(* Logix 5000 project; controller PLCbox vendor 1 type 14 code 149 rev 30.11; software revision 30.01; part 2 of 3 *)
(* tags used below, declared in another part *)
   HMI_Int_BOOL : BOOL[64];
   Light1_Complete_ONS : BOOL;
   Light1_Green : BOOL;
   Light1_Green_T : TIMER;
   Light1_Red : BOOL;
   Light1_Reset : BOOL;
   Light1_Yellow : BOOL;
   Light1_Yellow_T : TIMER;
   Light2_Complete_ONS : BOOL;
   Light2_Green : BOOL;
   Light2_Green_T : TIMER;
   Light2_Red : BOOL;
   Light2_Reset : BOOL;
   Light2_Yellow : BOOL;
   Light2_Yellow_T : TIMER;
   PID_Analog_In : REAL[20];
   System_Timer : TIMER[100];
   tagToPi : DINT;

PROGRAM MainProgram2   (* main routine _01_Main *)
VAR
   PID_1001 : PID_ENHANCED := (PVEUMax := 100.0, SPOper := 50.0, SPHLimit := 100.0, RatioProg := 1.0, RatioOper := 1.0, RatioHLimit := 1.0, RatioLLimit := 1.0, CVOper := 100.0, CVEUMax := 100.0, CVHLimit := 100.0, DependIndepend := 1, PGain := 0.1, IGain := 0.001, DGain := 0.001, PVEDerivative := 1, ProgOperReq := 1, RTSTime := 1, CVEU := 100.0, CV := 100.0, CVHAlarm := 1, SP := 50.0, SPPercent := 50.0, E := 50.0, EPercent := 50.0, InitPrimary := 1, WindupHOut := 1, Ratio := 1.0, Auto := 1, DeltaT := 0.1);
   PID_Par_1001 : UDT_PID := (P := 0.1, I := 0.001, D := 0.001, CV := 100.0, SP := 50.0, Auto := 1, Name := 'PID 1001 - Testing CLICK PLC Input');
   SCL_01 : SCALE := (InRawMax := 5000.0, InEUMax := 100.0);
END_VAR

ROUTINE _01_Main   (* ladder *)
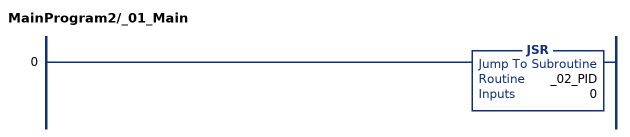
   0: JSR(_02_PID,0);
END_ROUTINE

ROUTINE _02_PID   (* function block diagram *)
   SHEET 1
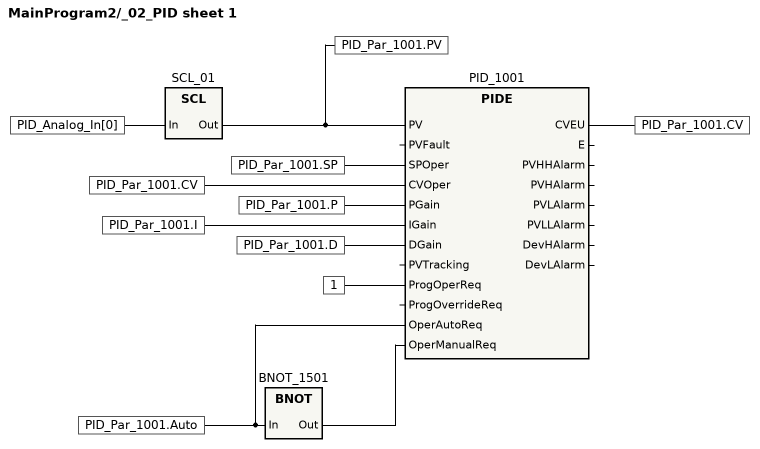
   SCL_01 : SCL(In := PID_Analog_In[0]);
   BNOT_1501 : BNOT(In := PID_Par_1001.Auto);
   PID_Par_1001.PV := SCL_01.Out;
   PID_1001 : PIDE(PV := SCL_01.Out, SPOper := PID_Par_1001.SP, CVOper := PID_Par_1001.CV, PGain := PID_Par_1001.P, IGain := PID_Par_1001.I, DGain := PID_Par_1001.D, ProgOperReq := 1, OperAutoReq := PID_Par_1001.Auto, OperManualReq := BNOT_1501.Out);   // unwired pins: PVFault PVTracking ProgOverrideReq E PVHHAlarm PVHAlarm PVLAlarm PVLLAlarm DevHAlarm DevLAlarm
   PID_Par_1001.CV := PID_1001.CVEU;
END_ROUTINE
END_PROGRAM

PROGRAM Mathematical   (* main routine _01_Main *)
VAR
   System_DINT : DINT[100] := ([0] := 12, [1] := 32, [2] := 54, [3] := 4, [4] := 31, [5] := 38, [6] := 100, [7] := 50, [8] := 200, [9] := 116);
   System_REAL : REAL[100] := ([0] := 23.0, [1] := 42.0, [2] := 0.48835304, [5] := 1.0);
END_VAR

ROUTINE _01_Main   (* ladder *)
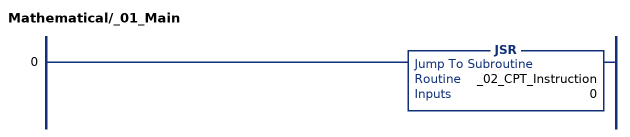
   0: JSR(_02_CPT_Instruction,0);
END_ROUTINE

ROUTINE _02_CPT_Instruction   (* ladder *)
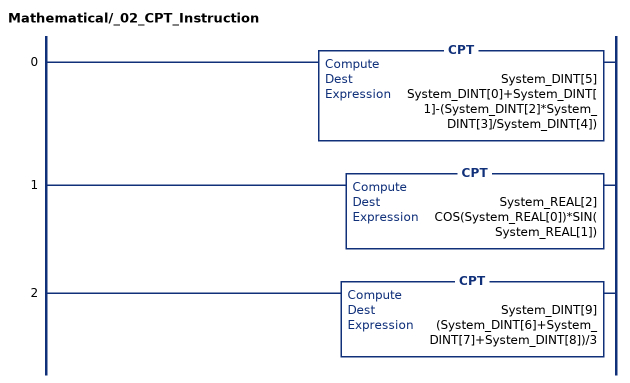
   0: CPT(System_DINT[5],System_DINT[0]+System_DINT[1]-(System_DINT[2]*System_DINT[3]/System_DINT[4]));
   1: CPT(System_REAL[2],COS(System_REAL[0])*SIN(System_REAL[1]));
   2: CPT(System_DINT[9],(System_DINT[6]+System_DINT[7]+System_DINT[8])/3);
END_ROUTINE
END_PROGRAM

PROGRAM PowerFlex525Mastery   (* main routine _01_Main *)
VAR
   Drive_Status : DINT := 1;
   Motor_Dev : REAL := 300.0;
   Motor_Fault_Timer : TIMER := (PRE := 20000);
   Motor_Faulted : BOOL;
   Motor_Run : BOOL;
   Motor_SpdLim_High : REAL := 6300.0;
   Motor_SpdLim_Low : REAL := 5700.0;
   Motor_Target_Speed_Fault : BOOL;
   Reset_PB : BOOL;
   Start_PB : BOOL;
   Stop_PB : BOOL;
END_VAR

ROUTINE _01_Main   (* ladder *)
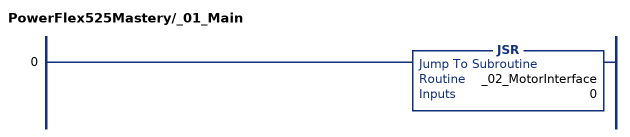
   0: JSR(_02_MotorInterface,0);
END_ROUTINE

ROUTINE _02_MotorInterface   (* ladder *)
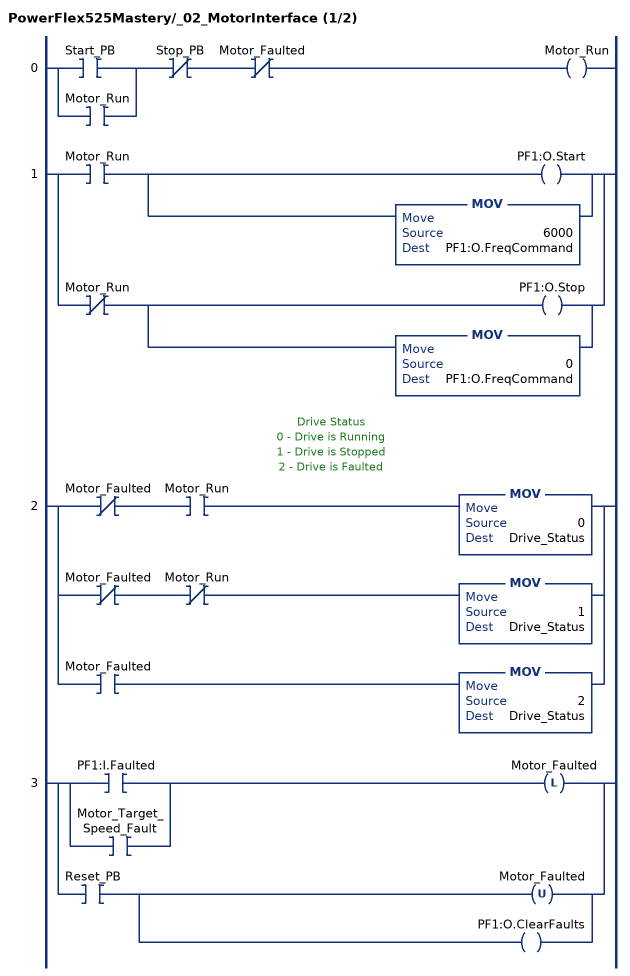
   0: [XIC(Start_PB) ,XIC(Motor_Run) ]XIO(Stop_PB)XIO(Motor_Faulted)OTE(Motor_Run);
   1: [XIC(Motor_Run) [OTE(PF1:O.Start) ,MOV(6000,PF1:O.FreqCommand) ] ,XIO(Motor_Run) [OTE(PF1:O.Stop) ,MOV(0,PF1:O.FreqCommand) ] ];
   // Drive Status
   // 0 - Drive is Running
   // 1 - Drive is Stopped
   // 2 - Drive is Faulted
   2: [XIO(Motor_Faulted) XIC(Motor_Run) MOV(0,Drive_Status) ,XIO(Motor_Faulted) XIO(Motor_Run) MOV(1,Drive_Status) ,XIC(Motor_Faulted) MOV(2,Drive_Status) ];
   3: [[XIC(PF1:I.Faulted) ,XIC(Motor_Target_Speed_Fault) ] OTL(Motor_Faulted) ,XIC(Reset_PB) [OTU(Motor_Faulted) ,OTE(PF1:O.ClearFaults) ] ];
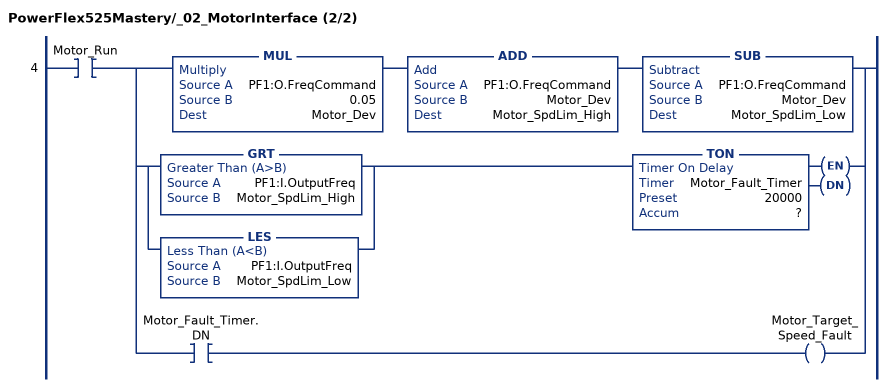
   4: XIC(Motor_Run)[MUL(PF1:O.FreqCommand,0.05,Motor_Dev) ADD(PF1:O.FreqCommand,Motor_Dev,Motor_SpdLim_High) SUB(PF1:O.FreqCommand,Motor_Dev,Motor_SpdLim_Low) ,[GRT(PF1:I.OutputFreq,Motor_SpdLim_High) ,LES(PF1:I.OutputFreq,Motor_SpdLim_Low) ] TON(Motor_Fault_Timer,?,?) ,XIC(Motor_Fault_Timer.DN) OTE(Motor_Target_Speed_Fault) ];
END_ROUTINE
END_PROGRAM

PROGRAM ST_Practice   (* main routine _01_Main *)

ROUTINE _01_Main   (* ladder *)
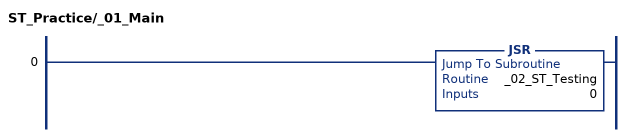
   0: JSR(_02_ST_Testing,0);
END_ROUTINE

ROUTINE _02_ST_Testing   (* structured text *)
   
END_ROUTINE
END_PROGRAM

PROGRAM StreetLightSystem   (* main routine _01_Main *)

ROUTINE _01_Main   (* ladder *)
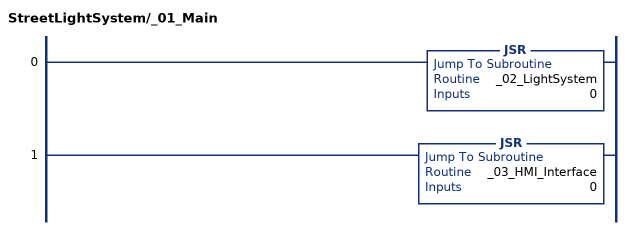
   0: JSR(_02_LightSystem,0);
   1: JSR(_03_HMI_Interface,0);
END_ROUTINE

ROUTINE _02_LightSystem   (* ladder *)
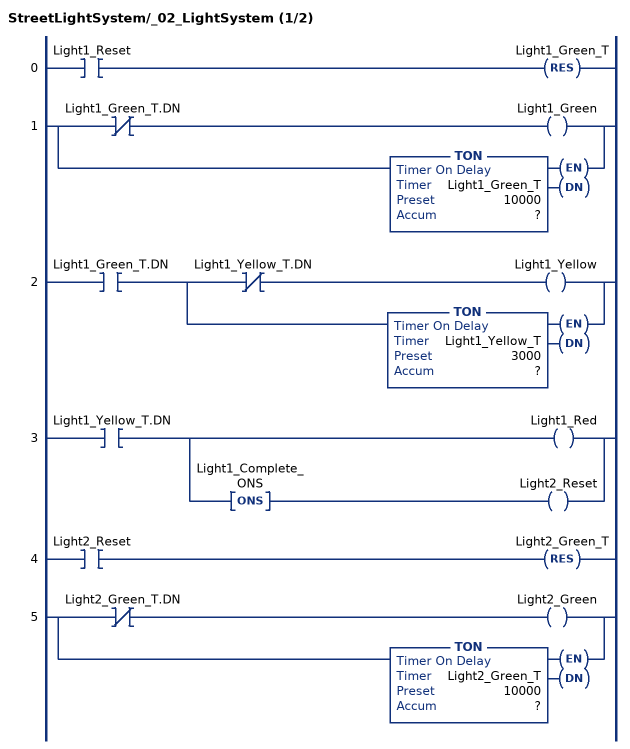
   0: XIC(Light1_Reset)RES(Light1_Green_T);
   1: [XIO(Light1_Green_T.DN) OTE(Light1_Green) ,TON(Light1_Green_T,?,?) ];
   2: XIC(Light1_Green_T.DN)[XIO(Light1_Yellow_T.DN) OTE(Light1_Yellow) ,TON(Light1_Yellow_T,?,?) ];
   3: XIC(Light1_Yellow_T.DN)[OTE(Light1_Red) ,ONS(Light1_Complete_ONS) OTE(Light2_Reset) ];
   4: XIC(Light2_Reset)RES(Light2_Green_T);
   5: [XIO(Light2_Green_T.DN) OTE(Light2_Green) ,TON(Light2_Green_T,?,?) ];
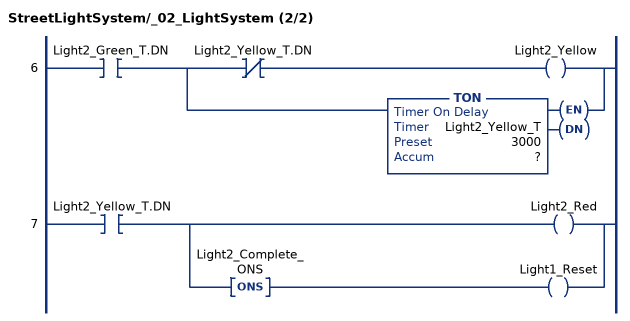
   6: XIC(Light2_Green_T.DN)[XIO(Light2_Yellow_T.DN) OTE(Light2_Yellow) ,TON(Light2_Yellow_T,?,?) ];
   7: XIC(Light2_Yellow_T.DN)[OTE(Light2_Red) ,ONS(Light2_Complete_ONS) OTE(Light1_Reset) ];
END_ROUTINE

ROUTINE _03_HMI_Interface   (* ladder *)
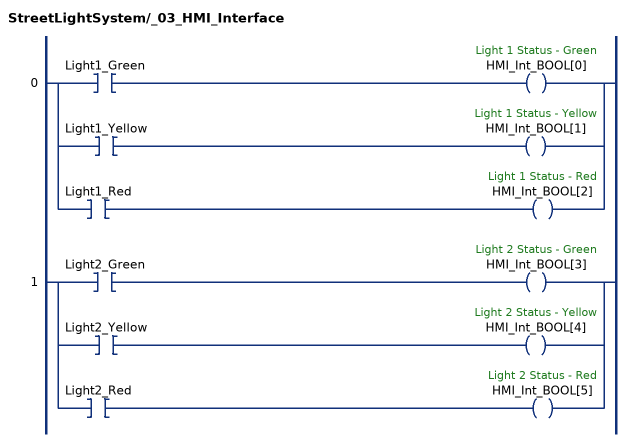
   0: [XIC(Light1_Green) OTE(HMI_Int_BOOL[0]) ,XIC(Light1_Yellow) OTE(HMI_Int_BOOL[1]) ,XIC(Light1_Red) OTE(HMI_Int_BOOL[2]) ];
   1: [XIC(Light2_Green) OTE(HMI_Int_BOOL[3]) ,XIC(Light2_Yellow) OTE(HMI_Int_BOOL[4]) ,XIC(Light2_Red) OTE(HMI_Int_BOOL[5]) ];
END_ROUTINE
END_PROGRAM

PROGRAM TankFillingChallenge   (* main routine _01_Main *)
VAR
   DischargeStatus : DINT := 1;
   FillingStatus : DINT := 1;
   T_Vlad : BOOL[128];
   TankActualLevel : REAL := 42.792046;
   TankDischargeRate : REAL := 0.5;
   TankEmptyThreshold : REAL := 5.0;
   TankFill : BOOL[128];
        [0]   // START Filling Station
        [1]   // STOP Filling Station
        [2]   // Filling Station RUNNING
        [3]   // START Discharge Station
        [4]   // STOP Discharge Station
        [5]   // Discharge Station RUNNING
        [6]   // TANK FULL
        [7]   // TANK EMPTY
   TankFillRate : REAL := 0.3;
   TankFullThreshold : REAL := 100.0;
   TankOut : BOOL[32];
        [0]   // Filling Station VALVE OPEN
        [1]   // Discharge Station VALVE OPEN
   TankTimers : TIMER[10] := ([0].PRE := 20, [1].PRE := 20);
END_VAR

ROUTINE _01_Main   (* ladder *)
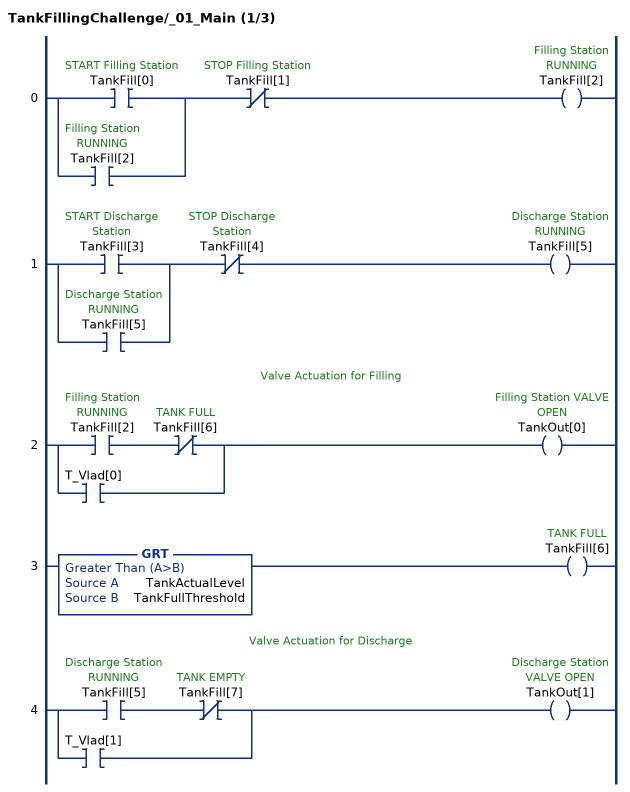
   0: [XIC(TankFill[0]) ,XIC(TankFill[2]) ]XIO(TankFill[1])OTE(TankFill[2]);
   1: [XIC(TankFill[3]) ,XIC(TankFill[5]) ]XIO(TankFill[4])OTE(TankFill[5]);
   // Valve Actuation for Filling
   2: [XIC(TankFill[2]) XIO(TankFill[6]) ,XIC(T_Vlad[0]) ]OTE(TankOut[0]);
   3: GRT(TankActualLevel,TankFullThreshold)OTE(TankFill[6]);
   // Valve Actuation for Discharge
   4: [XIC(TankFill[5]) XIO(TankFill[7]) ,XIC(T_Vlad[1]) ]OTE(TankOut[1]);
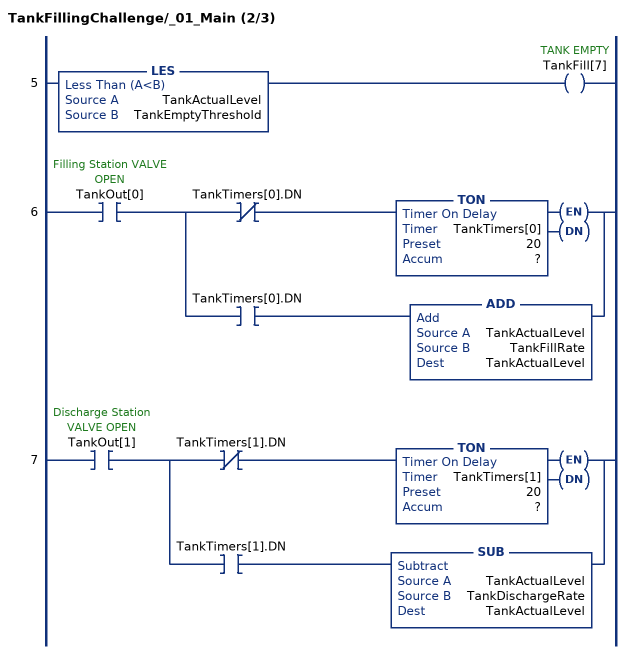
   5: LES(TankActualLevel,TankEmptyThreshold)OTE(TankFill[7]);
   6: XIC(TankOut[0])[XIO(TankTimers[0].DN) TON(TankTimers[0],?,?) ,XIC(TankTimers[0].DN) ADD(TankActualLevel,TankFillRate,TankActualLevel) ];
   7: XIC(TankOut[1])[XIO(TankTimers[1].DN) TON(TankTimers[1],?,?) ,XIC(TankTimers[1].DN) SUB(TankActualLevel,TankDischargeRate,TankActualLevel) ];
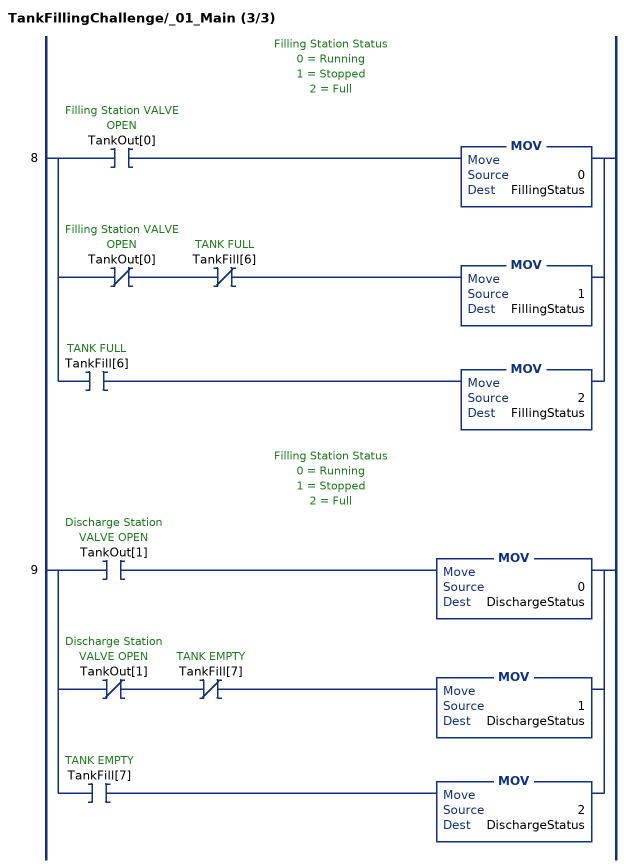
   // Filling Station Status
   // 0 = Running
   // 1 = Stopped
   // 2 = Full
   8: [XIC(TankOut[0]) MOV(0,FillingStatus) ,XIO(TankOut[0]) XIO(TankFill[6]) MOV(1,FillingStatus) ,XIC(TankFill[6]) MOV(2,FillingStatus) ];
   // Filling Station Status
   // 0 = Running
   // 1 = Stopped
   // 2 = Full
   9: [XIC(TankOut[1]) MOV(0,DischargeStatus) ,XIO(TankOut[1]) XIO(TankFill[7]) MOV(1,DischargeStatus) ,XIC(TankFill[7]) MOV(2,DischargeStatus) ];
END_ROUTINE
END_PROGRAM

PROGRAM TestProgram   (* main routine Main *)
VAR
   ALARM : BOOL[256];
   ALARM2 : BOOL[256];
   ALARM_DESC : String20;
   ALARM_DESCR : String20[256] := ([0] := 'Fault 0', [1] := 'Fault 1', [2] := 'Fault 2');
   EmptyString : String20;
   FaultDesc : String20 := 'Fault 1';
   FaultDesc2 : String20 := 'Fault 1';
   HMI_BOOL : BOOL[32];
   Index : DINT := 256;
   PLC_BOOL : BOOL[32];
   System_Cond : BOOL[256] := ([0] := 1);
        [0]   // Start MOTOR 1
        [1]   // MOTOR 1 At Target Speed
        [2]   // Start MOTOR 2
        [3]   // Motor 2 at Target Speed
        [4]   // Heat Boiler
        [5]   // Boiler at Temp
        [6]   // System Running
        [7]   // System FAULTED
        [8]   // System RESET
   System_INT : INT[10] := ([0] := 456, [1] := 456, [2] := 1);
   System_REAL : REAL[10] := ([0] := 54.0, [1] := 54.0, [2] := 54.0);
   System_STR : STRING[10];
   System_STRING : String20[10];
   SystemFaulted : BOOL := 1;
   SystemFaulted2 : BOOL := 1;
   SystemStart : BOOL;
   SytemReset : BOOL;
   SytemReset2 : BOOL;
END_VAR

ROUTINE _02_MOV_Instruction   (* ladder *)
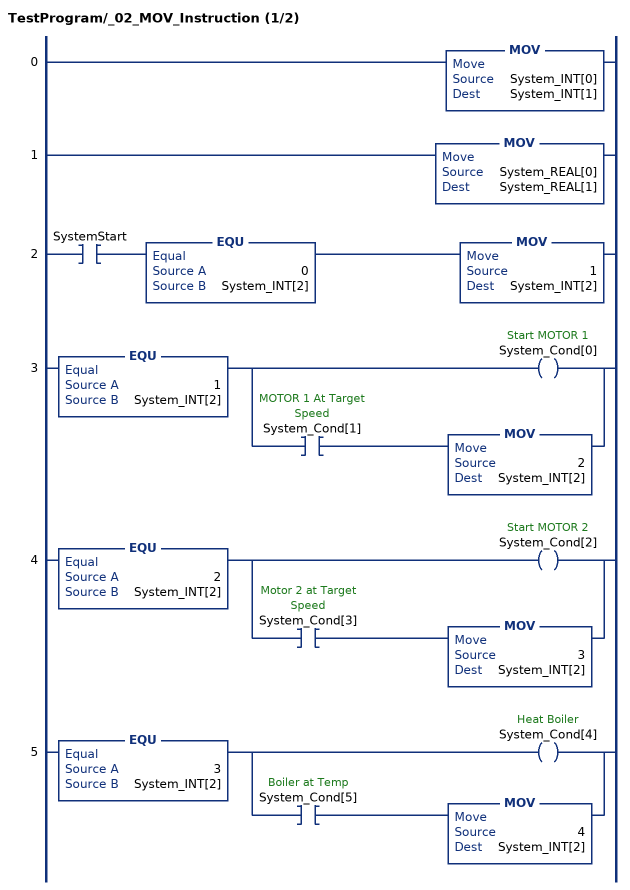
   0: MOV(System_INT[0],System_INT[1]);
   1: MOV(System_REAL[0],System_REAL[1]);
   2: XIC(SystemStart)EQU(0,System_INT[2])MOV(1,System_INT[2]);
   3: EQU(1,System_INT[2])[OTE(System_Cond[0]) ,XIC(System_Cond[1]) MOV(2,System_INT[2]) ];
   4: EQU(2,System_INT[2])[OTE(System_Cond[2]) ,XIC(System_Cond[3]) MOV(3,System_INT[2]) ];
   5: EQU(3,System_INT[2])[OTE(System_Cond[4]) ,XIC(System_Cond[5]) MOV(4,System_INT[2]) ];
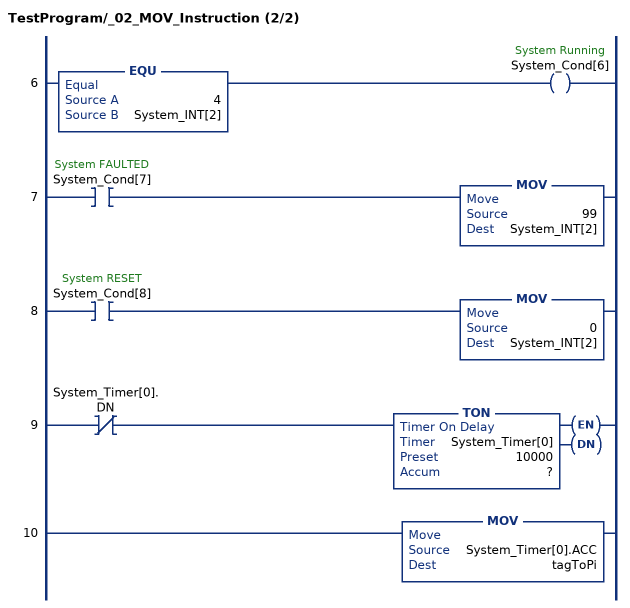
   6: EQU(4,System_INT[2])OTE(System_Cond[6]);
   7: XIC(System_Cond[7])MOV(99,System_INT[2]);
   8: XIC(System_Cond[8])MOV(0,System_INT[2]);
   9: XIO(System_Timer[0].DN)TON(System_Timer[0],?,?);
   10: MOV(System_Timer[0].ACC,tagToPi);
END_ROUTINE

ROUTINE _03_HMI   (* ladder *)
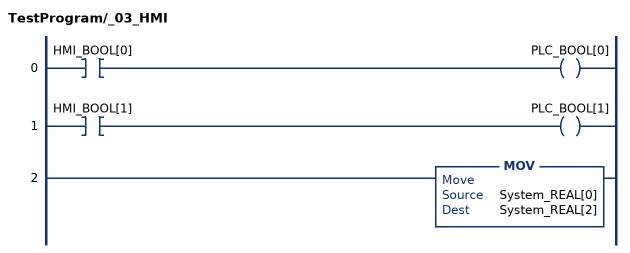
   0: XIC(HMI_BOOL[0])OTE(PLC_BOOL[0]);
   1: XIC(HMI_BOOL[1])OTE(PLC_BOOL[1]);
   2: MOV(System_REAL[0],System_REAL[2]);
END_ROUTINE
